(* PLC project codesysParallelTest.project, CODESYS CODESYS V3.5 SP17 Patch 3 *)
(* stored: creationDateTime 2022-12-11T22:12:58.0581928, modificationDateTime 2022-11-27T22:15:16.6542829 *)

PROGRAM PLC_PRG

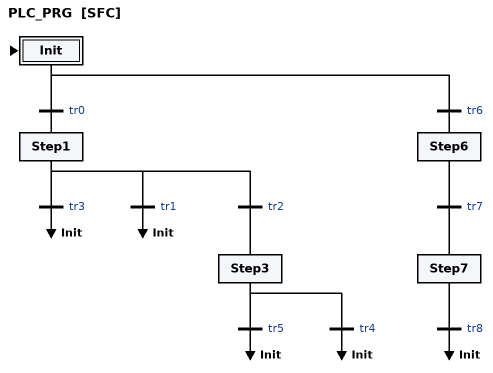
INITIAL_STEP Init:
END_STEP
TRANSITION FROM Init TO Step1
  := tr0;
END_TRANSITION
TRANSITION FROM Init TO Step6
  := tr6;
END_TRANSITION
STEP Step1:
END_STEP
TRANSITION FROM Step1 TO Init
  := tr3;
END_TRANSITION
TRANSITION FROM Step1 TO Init
  := tr1;
END_TRANSITION
TRANSITION FROM Step1 TO Step3
  := tr2;
END_TRANSITION
STEP Step3:
END_STEP
TRANSITION FROM Step3 TO Init
  := tr5;
END_TRANSITION
TRANSITION FROM Step3 TO Init
  := tr4;
END_TRANSITION
STEP Step6:
END_STEP
TRANSITION FROM Step6 TO Step7
  := tr7;
END_TRANSITION
STEP Step7:
END_STEP
TRANSITION FROM Step7 TO Init
  := tr8;
END_TRANSITION
END_PROGRAM
